SUBAPPLICATION Ventilsteuerung_Uebung_001_P2 (* DigitalInput_I1 auf DigitalOutput_Q1, mit Plug and Socket *)
  (* Standard: 61499-2 *)
  (* Version 1.0, 2023-10-23, franz *)
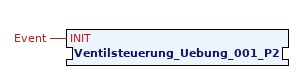
  EVENT_INPUT
    INIT;
  END_EVENT
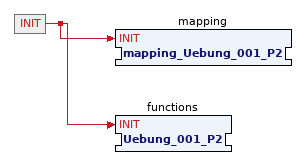
  SUBAPPS
    mapping : mapping_Uebung_001_P2;
    functions : Uebung_001_P2;
  END_SUBAPPS
  EVENT_CONNECTIONS
    INIT TO mapping.INIT;
    INIT TO functions.INIT;
  END_CONNECTIONS
END_SUBAPPLICATION
